{attribute 'qualified_only'}
{attribute 'strict'}
{attribute 'to_string'}
TYPE AktorStatus :
(
	default := 0,
	inRP,
	inAP,
	
	zuRP,
	zuAP
);
END_TYPE

(* stored: Version 1.1.0.1, ProductVersion 3.1.4024.12
   DUT AktorStatus: Id {cddc2ffb-e141-4e0b-834b-0b45c595cd86} *)
